// TIA Portal project "Multi DQ" (V17)

(* hardware
DEVICE "S7-1200 station_1"  S7-1200 Station
   slot 0: "Rack_0"  S7-1200 Rack  Rack  V1.0
   slot 1: "Hello_World"  CPU 1214C DC/DC/DC  6ES7 214-1AG40-0XB0  V4.5
*)

// ===== PLC "Hello_World"  CPU 1214C DC/DC/DC =====

VAR_GLOBAL   // PLC tag table "Default tag table"
   "Blue_Light" AT %Q0.0 : Bool;
   "Stop button (NC)" AT %I0.0 : Bool;
   "Red_Light" AT %Q0.4 : Bool;
   "Yellow_Light" AT %Q0.5 : Bool;
   "Green_Light" AT %Q0.6 : Bool;
   "White_Light" AT %Q0.7 : Bool;
   "AlwaysTRUE" AT %M1.2 : Bool;
   "AlwaysFALSE" AT %M1.3 : Bool;
   "Clock_Byte" AT %MB0 : Byte;
   "Clock_10Hz" AT %M0.0 : Bool;
   "Clock_5Hz" AT %M0.1 : Bool;
   "Clock_2.5Hz" AT %M0.2 : Bool;
   "Clock_2Hz" AT %M0.3 : Bool;
   "Clock_1.25Hz" AT %M0.4 : Bool;
   "Clock_1Hz" AT %M0.5 : Bool;
   "Clock_0.625Hz" AT %M0.6 : Bool;
   "Clock_0.5Hz" AT %M0.7 : Bool;
   "SR01" AT %M2.0 : Bool;
   "Reset_up" AT %M2.1 : Bool;
   "System_Byte" AT %MB1 : Byte;
   "Start Button" AT %I0.1 : Bool;
   "Buzzer" AT %Q1.1 : Bool;
END_VAR

DATA_BLOCK "Passthrough_DB"   // DB1
{ S7_Optimized_Access := 'TRUE' }
VERSION : 0.1
// stored: InstanceOfName Passthrough
"Passthrough"
BEGIN
END_DATA_BLOCK

// folder: System blocks/Program resources

DATA_BLOCK "IEC_Counter_0_DB"   // DB2
{ S7_Optimized_Access := 'TRUE' }
AUTHOR : Simatic
FAMILY : IEC
NAME : CNTR
VERSION : 1.0
// stored: InstanceOfName IEC_COUNTER
"IEC_COUNTER"
BEGIN
END_DATA_BLOCK

// folder: (top level)

FUNCTION_BLOCK "Passthrough"   // FB1, LAD
{ S7_Optimized_Access := 'TRUE' }
VERSION : 0.1
   VAR_INPUT
      IN : Bool;
      MAX_COUNT : Int;
   END_VAR
   VAR_OUTPUT
      PASS_1 : Bool;
      PASS_2 : Bool;
      PASS_3 : Bool;
      "NOT" : Bool;
      COUNT : Int;
      BUZZER : Bool;
   END_VAR
   VAR_TEMP
      MAX_COUNT_REACH : Bool;
   END_VAR
   VAR_TEMP   // added for the SCL form of the ladder/FBD networks
      _w1 : Bool;
   END_VAR
BEGIN

REGION Network 1
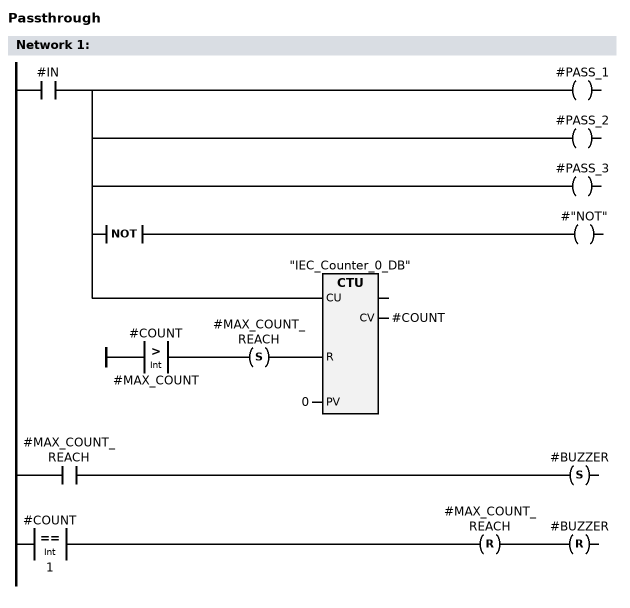
   #PASS_1 := #IN;
   #PASS_2 := #IN;
   #PASS_3 := #IN;
   #"NOT" := NOT #IN;
   #_w1 := #COUNT > #MAX_COUNT;
   IF #_w1 THEN #MAX_COUNT_REACH := TRUE; END_IF;
   "IEC_Counter_0_DB".CTU(CU := #IN, R := #_w1, PV := 0, CV => #COUNT);
   IF #MAX_COUNT_REACH THEN #BUZZER := TRUE; END_IF;
   IF #COUNT = 1 THEN
       #MAX_COUNT_REACH := FALSE;
       #BUZZER := FALSE;
   END_IF;
END_REGION
END_FUNCTION_BLOCK

ORGANIZATION_BLOCK "Main"   // OB1, LAD, ProgramCycle
TITLE = "Main Program Sweep (Cycle)"
{ S7_Optimized_Access := 'TRUE' }
VERSION : 0.1
   VAR_INPUT
      Initial_Call : Bool;   // Initial call of this OB
      Remanence : Bool;   // =True, if remanent data are available
   END_VAR
   VAR_TEMP   // added for the SCL form of the ladder/FBD networks
      _w1 : Bool;
   END_VAR
BEGIN

REGION Network 1
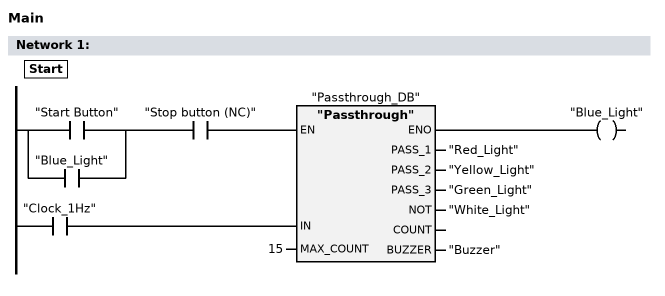
   Label( Start )
   RUNG wire#powerrail
      Contact( "Start Button" )
      wire#w1
      Contact( "Stop button (NC)" )
      "Passthrough_DB"(IN := wire#w2, MAX_COUNT := 15, PASS_1 => "Red_Light", PASS_2 => "Yellow_Light", PASS_3 => "Green_Light", "NOT" => "White_Light", COUNT =>, BUZZER => "Buzzer")
      Coil( "Blue_Light" )
   END_RUNG
   RUNG wire#powerrail
      Contact( "Blue_Light" )
   END_RUNG wire#w1
   RUNG wire#powerrail
      Contact( "Clock_1Hz" )
   END_RUNG wire#w2
   // the same network as SCL:
   Start:
   "Passthrough_DB"(EN := ("Start Button" OR "Blue_Light") AND "Stop button (NC)",   // "Passthrough"
                    IN := "Clock_1Hz",
                    MAX_COUNT := 15,
                    PASS_1 => "Red_Light",
                    PASS_2 => "Yellow_Light",
                    PASS_3 => "Green_Light",
                    "NOT" => "White_Light",
                    BUZZER => "Buzzer",
                    ENO => #_w1);
   "Blue_Light" := #_w1;
END_REGION
END_ORGANIZATION_BLOCK